Universal Robots PolyScope program: tvt19spl_unload_8.urp

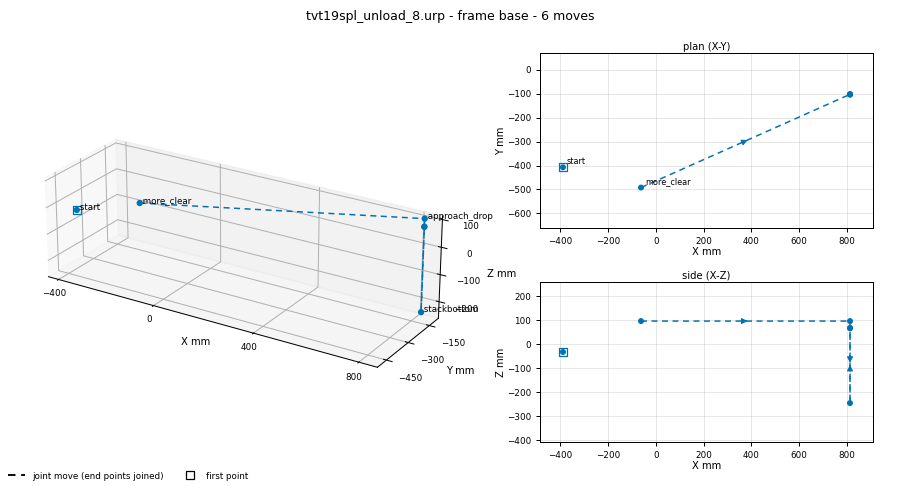
[picture p0: tool path of tvt19spl_unload_8.urp in frame base, 6 of 10 moves have a stored position in this frame; points joined in program order, loops and branches not executed]
Program tvt19spl_unload_8 (installation=default directory=/programs/usbdisk/TVT19SPL createdIn=3.15.4.106291 lastSavedIn=3.15.4.106291 robotSerialNumber=2018357902)
Calibrated DH parameters: a=[0.00015, -0.193406, -0.353214, 0.000101, 0.000049, 0]; d=[0.08934, 486.592682, -461.422552, -25.060198, 0.094902, 0.082419]; alpha=[1.570675, -0.000778, -0.00678, 1.570332, -1.570641, 0]; deltaTheta=[0.000035, -1.098336, 0.64827, 0.450067, -0.000055, 0.000056]
BeforeStart
  Folder Before the beginning
    URCap Gripper Activate (Robotiq_Grippers, Robotiq Inc.) dataModel(ResetAndActivateKey=false)
    URCap Gripper (Robotiq_Grippers, Robotiq Inc.) dataModel(position=0.0, force=0.0, speed=0.0, positionInDouble=0.0, forceInDouble=0.0, speedInDouble=0.0, slaveIds=[9], blocking=true)
    eka_auto := True
    'Connect to the control device'
    pcip := "192.168.100.5"
    connection1 := False
    Loop While (checkContinuously=false) expression=connection1≟ False
      connection1 := socket_open(pcip,1201)
Robot Program (runOnlyOnce=false)
  'Receive order'
  orders := socket_read_string(timeout=0)
  If orders ≟ "first"
    eka_auto := True
  MoveJ speed 150 deg/s, acceleration 120 deg/s^2 (useActiveTCP=true)
    Waypoint start: TCP in base x=-387.858 y=-407.223 z=-32.068 mm, rx=-0.0001 ry=-3.0439 rz=0.7772 rad; joints [-130.25, -112.975, -123.602, -10.932, 108.111, -37.045] deg; flange x=-387.854 y=-325.72 z=117.122 mm, rx=-0.0001 ry=-3.0439 rz=0.7772 rad
  'look for a inbound car'
